(* Logix 5000 project; controller R5_CSS vendor 1 type 14 code 74 rev 19.11; software revision 19.01; part 19 of 20 *)
(* tags used below, declared in another part *)
   AlarmMasterDisable : BOOL;
   AutoTune : PIDE_AUTOTUNE;
   CSS_Heartbeat : BOOL;
   CSS_HeartbeatOffONS : BOOL;
   CSS_HeartbeatOnONS : BOOL;
   CSS_OK_TO_RUN : BOOL;   // PRU_RUN_DISABLE 0 = Cannot Run 1 = OK to Run
   CSS_Status_To_UTL_Comms : DINT;
   Fault : BOOL;
   FC101 : FLOW_CONTROL;   // QUENCH BASIN FLOW TRANSMITTER CONTROL
   FC101_Initialize : BOOL;
   FC101_Initialize_TON : TIMER;
   FT140_TOTAL_FLOW : REAL;
   LC101 : LEVEL_CONTROL;   // QUENCH TOWER BASIN LIT
   LC101_PIDE_AUTO : BOOL;
   LC101_PIDE_CV_Hold : REAL;
   LC303A : LEVEL_CONTROL;   // AQUEOUS PHASE OF PRIMARY SETTLER
   MSG_ConnectionRateSec : DINT;
   MSG_TimeoutMultiplier : DINT;
   MSG_UnconnectedTimeoutSec : DINT;
   PRU_Batch_Start : BOOL[32];
   PRU_Batch_Stop : BOOL[32];
   PRU_BatchNewID : DINT[10];
   PRU_BLOWER_SEQ : INT;   // PRU BLOWER SEQUENCE NUMBER
   PRU_MSG_CommsPath : MSG_CommsPath[9];
   PRU_MSG_Prefix : STRING;
   PRU_Quantity : DINT;
   PRU_SEQ_TMR : TIMER;   // PRU_SEQUENCE TIMER
   PRUA_Batch_Start_ONS : BOOL;
   PRUA_Batch_Stop_ONS : BOOL;
   PRUA_READ : INT[30];
   PRUA_READ_MSG : MESSAGE;
   PRUA_WRITE_MSG : MESSAGE;
   PRUB_Batch_Start_ONS : BOOL;
   PRUB_Batch_Stop_ONS : BOOL;
   PRUB_READ : INT[30];
   PRUB_READ_MSG : MESSAGE;
   PRUB_WRITE_MSG : MESSAGE;
   PRUC_Batch_Start_ONS : BOOL;
   PRUC_Batch_Stop_ONS : BOOL;
   PRUC_READ : INT[30];
   PRUC_READ_MSG : MESSAGE;
   PRUC_WRITE_MSG : MESSAGE;
   PRUD_Batch_Start_ONS : BOOL;
   PRUD_Batch_Stop_ONS : BOOL;
   PRUD_READ : INT[30];   // PRU D READ
   PRUD_READ_MSG : MESSAGE;
   PRUD_WRITE_MSG : MESSAGE;
   PRUE_Batch_Start_ONS : BOOL;
   PRUE_Batch_Stop_ONS : BOOL;
   PRUE_READ : INT[30];
   PRUE_READ_MSG : MESSAGE;
   PRUE_WRITE_MSG : MESSAGE;
   PRUF_Batch_Start_ONS : BOOL;
   PRUF_Batch_Stop_ONS : BOOL;
   PRUF_READ : INT[30];
   PRUF_READ_MSG : MESSAGE;
   PRUF_WRITE_MSG : MESSAGE;
   PRUG_Batch_Start_ONS : BOOL;
   PRUG_Batch_Stop_ONS : BOOL;
   PRUG_READ : INT[30];
   PRUG_READ_MSG : MESSAGE;
   PRUG_WRITE_MSG : MESSAGE;
   PRUH_Batch_Start_ONS : BOOL;
   PRUH_Batch_Stop_ONS : BOOL;
   PRUH_READ : INT[30];
   PRUH_READ_MSG : MESSAGE;
   PRUH_WRITE_MSG : MESSAGE;
   TestyBit : DINT;
   UTIL_1 : INT;   // ONE SHOTS FOR UTILITIES
   UTL_AlarmMaster : DINT;
   UTL_Comms : DINT[3];
   UTL_CommsLossAlm : BOOL;
   UTL_HeartbeatTimer : TIMER;
   UTL_READ_MSG : MESSAGE;
   WRS_OK : BOOL;
(* MainProgram, continued *)

ROUTINE TEMPORARY   (* ladder *)
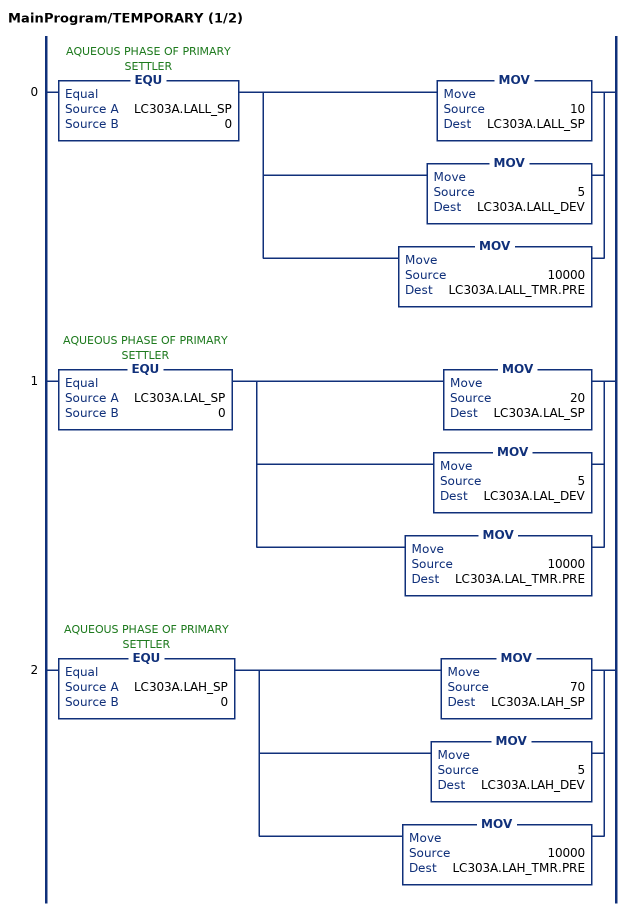
   0: EQU(LC303A.LALL_SP,0)[MOV(10,LC303A.LALL_SP) ,MOV(5,LC303A.LALL_DEV) ,MOV(10000,LC303A.LALL_TMR.PRE) ];
   1: EQU(LC303A.LAL_SP,0)[MOV(20,LC303A.LAL_SP) ,MOV(5,LC303A.LAL_DEV) ,MOV(10000,LC303A.LAL_TMR.PRE) ];
   2: EQU(LC303A.LAH_SP,0)[MOV(70,LC303A.LAH_SP) ,MOV(5,LC303A.LAH_DEV) ,MOV(10000,LC303A.LAH_TMR.PRE) ];
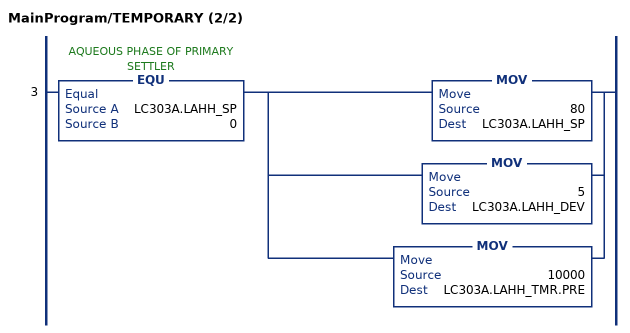
   3: EQU(LC303A.LAHH_SP,0)[MOV(80,LC303A.LAHH_SP) ,MOV(5,LC303A.LAHH_DEV) ,MOV(10000,LC303A.LAHH_TMR.PRE) ];
END_ROUTINE

ROUTINE UTIL   (* ladder *)
// UTILITIES LOGIC
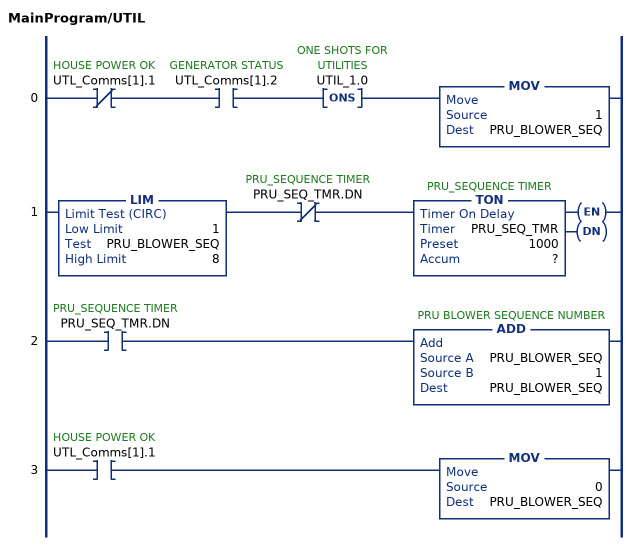
   0: XIO(UTL_Comms[1].1)XIC(UTL_Comms[1].2)ONS(UTIL_1.0)MOV(1,PRU_BLOWER_SEQ);
   1: LIM(1,PRU_BLOWER_SEQ,8)XIO(PRU_SEQ_TMR.DN)TON(PRU_SEQ_TMR,?,?);
   2: XIC(PRU_SEQ_TMR.DN)ADD(PRU_BLOWER_SEQ,1,PRU_BLOWER_SEQ);
   3: XIC(UTL_Comms[1].1)MOV(0,PRU_BLOWER_SEQ);
END_ROUTINE
END_PROGRAM

PROGRAM Never_Fault_Logic   (* main routine Main *)
VAR
   HMI_CONTROLLER_DISPLAY : MAJOR_FAULT := (TYPE := 3, CODE := 23);
   MAJORFAULT_RECORD : FAULTRECORD;
END_VAR

ROUTINE Main   (* ladder *)
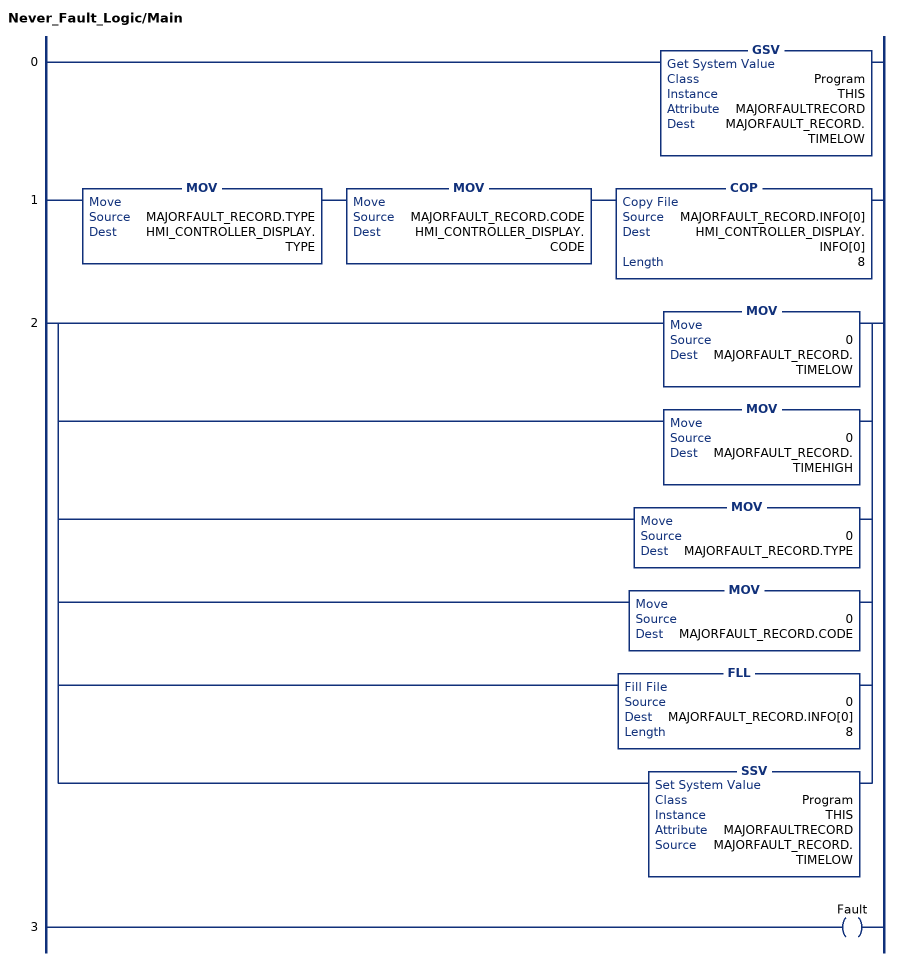
   0: GSV(Program,THIS,MAJORFAULTRECORD,MAJORFAULT_RECORD.TIMELOW);
   1: MOV(MAJORFAULT_RECORD.TYPE,HMI_CONTROLLER_DISPLAY.TYPE)MOV(MAJORFAULT_RECORD.CODE,HMI_CONTROLLER_DISPLAY.CODE)COP(MAJORFAULT_RECORD.INFO[0],HMI_CONTROLLER_DISPLAY.INFO[0],8);
   2: [MOV(0,MAJORFAULT_RECORD.TIMELOW) ,MOV(0,MAJORFAULT_RECORD.TIMEHIGH) ,MOV(0,MAJORFAULT_RECORD.TYPE) ,MOV(0,MAJORFAULT_RECORD.CODE) ,FLL(0,MAJORFAULT_RECORD.INFO[0],8) ,SSV(Program,THIS,MAJORFAULTRECORD,MAJORFAULT_RECORD.TIMELOW) ];
   3: OTE(Fault);
END_ROUTINE
END_PROGRAM

PROGRAM PIDE   (* main routine Main *)
VAR
   BNOT_01 : FBD_BOOLEAN_NOT := (Out := 1);
   BNOT_02 : FBD_BOOLEAN_NOT := (In := 1);
   SUB_01 : FBD_MATH := (SourceA := 1.4874992, SourceB := 30.0, Dest := -28.5125);
END_VAR

ROUTINE LC101   (* function block diagram *)
   SHEET 1
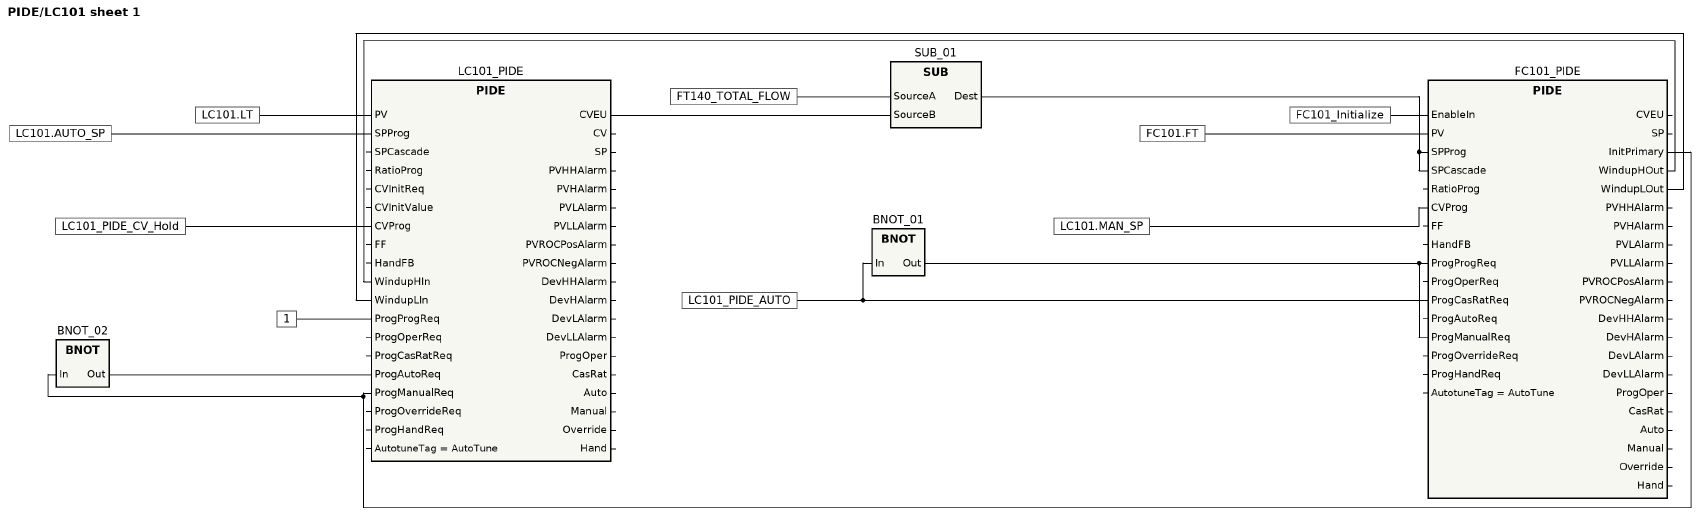
   BNOT_02 : BNOT(In := FC101_PIDE.InitPrimary {feedback});
   LC101_PIDE : PIDE(PV := LC101.LT, SPProg := LC101.AUTO_SP, CVProg := LC101_PIDE_CV_Hold, WindupHIn := FC101_PIDE.WindupHOut {feedback}, WindupLIn := FC101_PIDE.WindupLOut {feedback}, ProgProgReq := 1, ProgAutoReq := BNOT_02.Out, ProgManualReq := FC101_PIDE.InitPrimary {feedback}, AutotuneTag := AutoTune);   // unwired pins: SPCascade RatioProg CVInitReq CVInitValue FF HandFB ProgOperReq ProgCasRatReq ProgOverrideReq ProgHandReq CV SP PVHHAlarm PVHAlarm PVLAlarm PVLLAlarm PVROCPosAlarm PVROCNegAlarm DevHHAlarm DevHAlarm DevLAlarm DevLLAlarm ProgOper CasRat Auto Manual Override Hand
   BNOT_01 : BNOT(In := LC101_PIDE_AUTO);
   SUB_01 : SUB(SourceA := FT140_TOTAL_FLOW, SourceB := LC101_PIDE.CVEU);
   FC101_PIDE : PIDE(EnableIn := FC101_Initialize, PV := FC101.FT, SPProg := SUB_01.Dest, SPCascade := SUB_01.Dest, CVProg := LC101.MAN_SP, ProgProgReq := BNOT_01.Out, ProgCasRatReq := LC101_PIDE_AUTO, ProgManualReq := BNOT_01.Out, AutotuneTag := AutoTune);   // unwired pins: RatioProg FF HandFB ProgOperReq ProgAutoReq ProgOverrideReq ProgHandReq CVEU SP PVHHAlarm PVHAlarm PVLAlarm PVLLAlarm PVROCPosAlarm PVROCNegAlarm DevHHAlarm DevHAlarm DevLAlarm DevLLAlarm ProgOper CasRat Auto Manual Override Hand
END_ROUTINE

ROUTINE Main   (* ladder *)
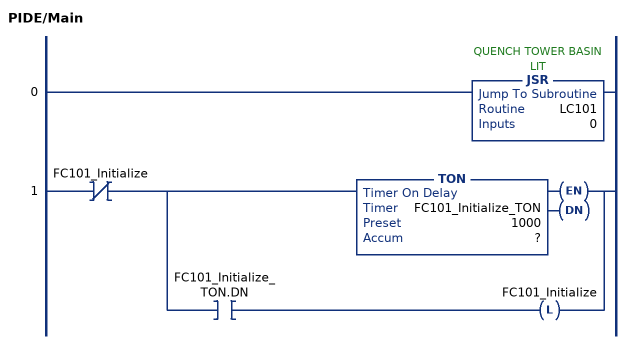
   0: JSR(LC101,0);
   1: XIO(FC101_Initialize)[TON(FC101_Initialize_TON,?,?) ,XIC(FC101_Initialize_TON.DN) OTL(FC101_Initialize) ];
END_ROUTINE
END_PROGRAM

PROGRAM POD1_MSG   (* main routine MSG *)
VAR
   PRU_BatchNewID_old : DINT[5];
END_VAR

ROUTINE MSG   (* ladder *)
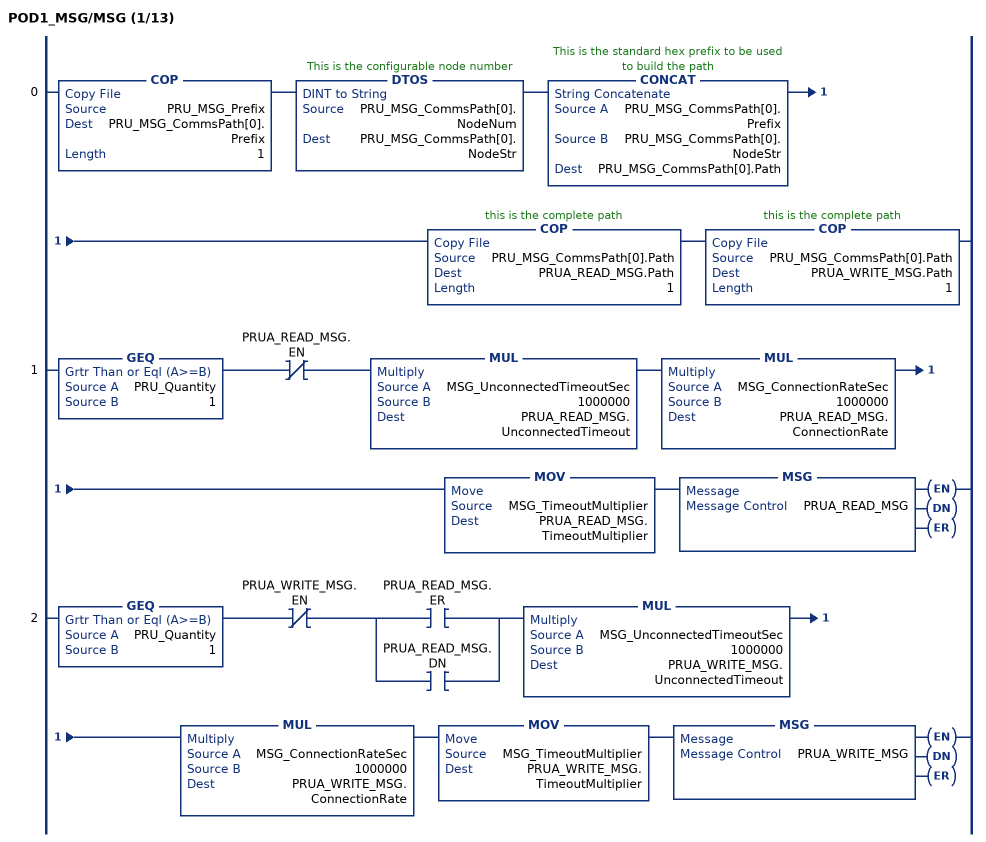
   0: COP(PRU_MSG_Prefix,PRU_MSG_CommsPath[0].Prefix,1)DTOS(PRU_MSG_CommsPath[0].NodeNum,PRU_MSG_CommsPath[0].NodeStr)CONCAT(PRU_MSG_CommsPath[0].Prefix,PRU_MSG_CommsPath[0].NodeStr,PRU_MSG_CommsPath[0].Path)COP(PRU_MSG_CommsPath[0].Path,PRUA_READ_MSG.Path,1)COP(PRU_MSG_CommsPath[0].Path,PRUA_WRITE_MSG.Path,1);
   1: GEQ(PRU_Quantity,1)XIO(PRUA_READ_MSG.EN)MUL(MSG_UnconnectedTimeoutSec,1000000,PRUA_READ_MSG.UnconnectedTimeout)MUL(MSG_ConnectionRateSec,1000000,PRUA_READ_MSG.ConnectionRate)MOV(MSG_TimeoutMultiplier,PRUA_READ_MSG.TimeoutMultiplier)MSG(PRUA_READ_MSG);
   2: GEQ(PRU_Quantity,1)XIO(PRUA_WRITE_MSG.EN)[XIC(PRUA_READ_MSG.ER) ,XIC(PRUA_READ_MSG.DN) ]MUL(MSG_UnconnectedTimeoutSec,1000000,PRUA_WRITE_MSG.UnconnectedTimeout)MUL(MSG_ConnectionRateSec,1000000,PRUA_WRITE_MSG.ConnectionRate)MOV(MSG_TimeoutMultiplier,PRUA_WRITE_MSG.TimeoutMultiplier)MSG(PRUA_WRITE_MSG);
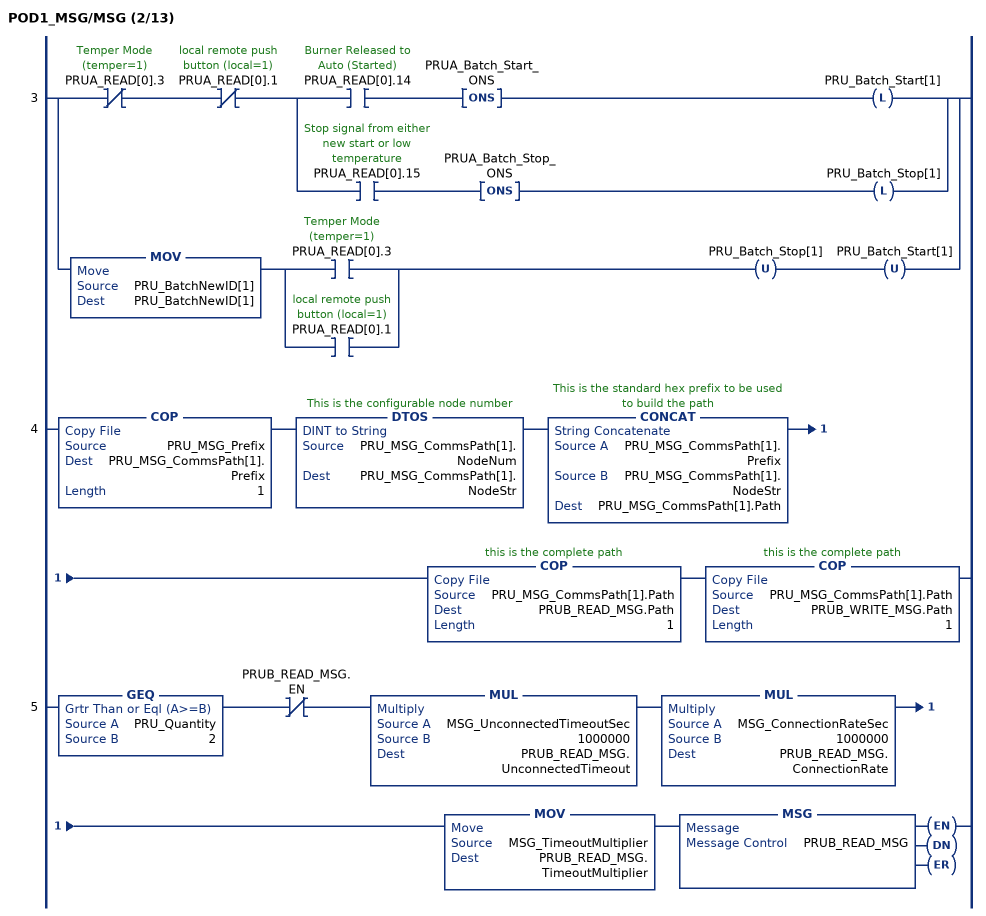
   3: [XIO(PRUA_READ[0].3) XIO(PRUA_READ[0].1) [XIC(PRUA_READ[0].14) ONS(PRUA_Batch_Start_ONS) OTL(PRU_Batch_Start[1]) ,XIC(PRUA_READ[0].15) ONS(PRUA_Batch_Stop_ONS) OTL(PRU_Batch_Stop[1]) ] ,MOV(PRU_BatchNewID[1],PRU_BatchNewID[1]) [XIC(PRUA_READ[0].3) ,XIC(PRUA_READ[0].1) ] OTU(PRU_Batch_Stop[1]) OTU(PRU_Batch_Start[1]) ];
   4: COP(PRU_MSG_Prefix,PRU_MSG_CommsPath[1].Prefix,1)DTOS(PRU_MSG_CommsPath[1].NodeNum,PRU_MSG_CommsPath[1].NodeStr)CONCAT(PRU_MSG_CommsPath[1].Prefix,PRU_MSG_CommsPath[1].NodeStr,PRU_MSG_CommsPath[1].Path)COP(PRU_MSG_CommsPath[1].Path,PRUB_READ_MSG.Path,1)COP(PRU_MSG_CommsPath[1].Path,PRUB_WRITE_MSG.Path,1);
   5: GEQ(PRU_Quantity,2)XIO(PRUB_READ_MSG.EN)MUL(MSG_UnconnectedTimeoutSec,1000000,PRUB_READ_MSG.UnconnectedTimeout)MUL(MSG_ConnectionRateSec,1000000,PRUB_READ_MSG.ConnectionRate)MOV(MSG_TimeoutMultiplier,PRUB_READ_MSG.TimeoutMultiplier)MSG(PRUB_READ_MSG);
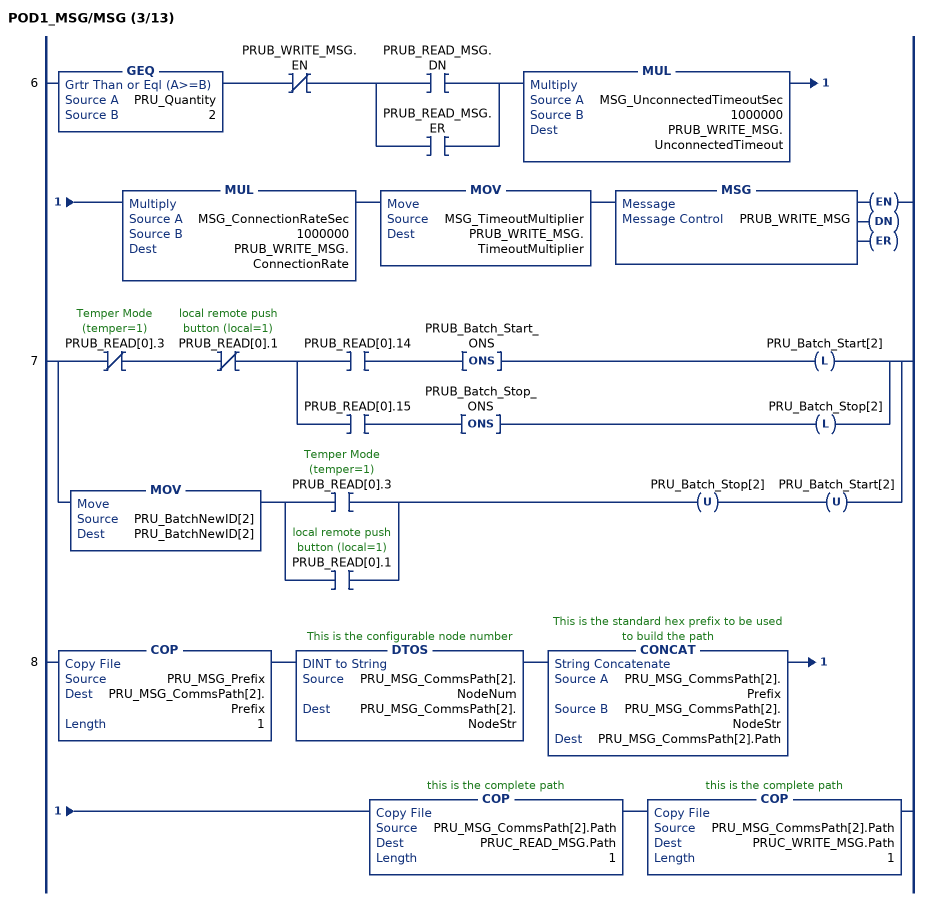
   6: GEQ(PRU_Quantity,2)XIO(PRUB_WRITE_MSG.EN)[XIC(PRUB_READ_MSG.DN) ,XIC(PRUB_READ_MSG.ER) ]MUL(MSG_UnconnectedTimeoutSec,1000000,PRUB_WRITE_MSG.UnconnectedTimeout)MUL(MSG_ConnectionRateSec,1000000,PRUB_WRITE_MSG.ConnectionRate)MOV(MSG_TimeoutMultiplier,PRUB_WRITE_MSG.TimeoutMultiplier)MSG(PRUB_WRITE_MSG);
   7: [XIO(PRUB_READ[0].3) XIO(PRUB_READ[0].1) [XIC(PRUB_READ[0].14) ONS(PRUB_Batch_Start_ONS) OTL(PRU_Batch_Start[2]) ,XIC(PRUB_READ[0].15) ONS(PRUB_Batch_Stop_ONS) OTL(PRU_Batch_Stop[2]) ] ,MOV(PRU_BatchNewID[2],PRU_BatchNewID[2]) [XIC(PRUB_READ[0].3) ,XIC(PRUB_READ[0].1) ] OTU(PRU_Batch_Stop[2]) OTU(PRU_Batch_Start[2]) ];
   8: COP(PRU_MSG_Prefix,PRU_MSG_CommsPath[2].Prefix,1)DTOS(PRU_MSG_CommsPath[2].NodeNum,PRU_MSG_CommsPath[2].NodeStr)CONCAT(PRU_MSG_CommsPath[2].Prefix,PRU_MSG_CommsPath[2].NodeStr,PRU_MSG_CommsPath[2].Path)COP(PRU_MSG_CommsPath[2].Path,PRUC_READ_MSG.Path,1)COP(PRU_MSG_CommsPath[2].Path,PRUC_WRITE_MSG.Path,1);
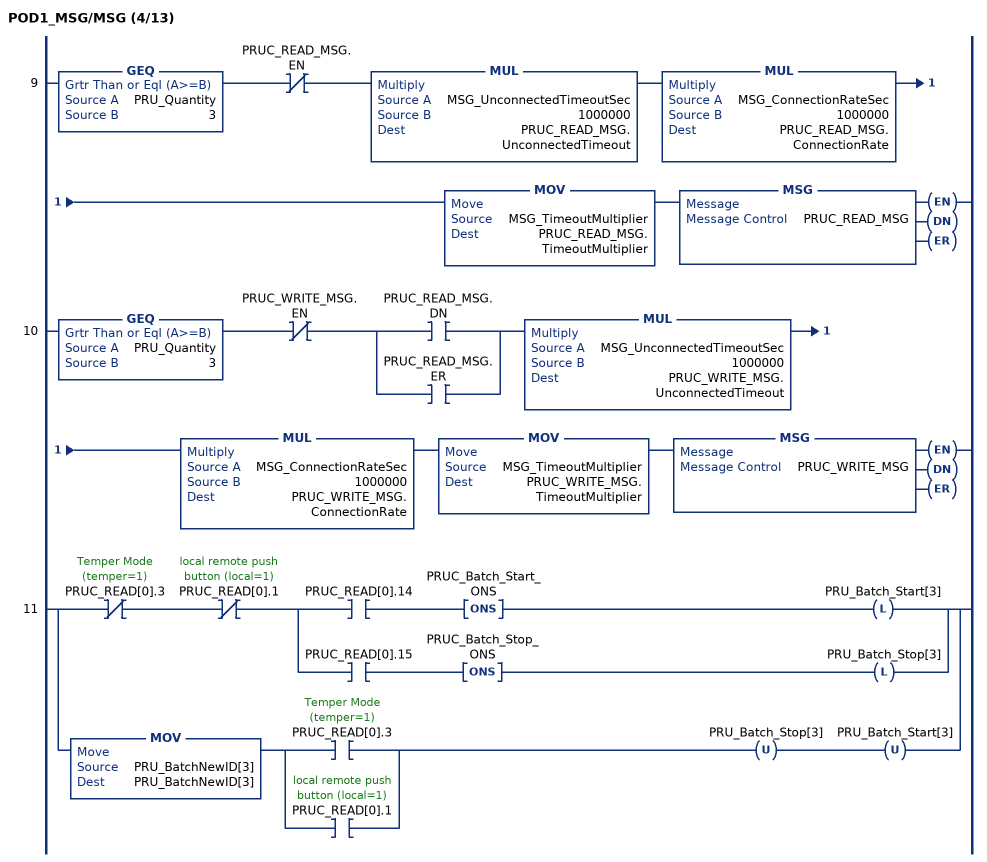
   9: GEQ(PRU_Quantity,3)XIO(PRUC_READ_MSG.EN)MUL(MSG_UnconnectedTimeoutSec,1000000,PRUC_READ_MSG.UnconnectedTimeout)MUL(MSG_ConnectionRateSec,1000000,PRUC_READ_MSG.ConnectionRate)MOV(MSG_TimeoutMultiplier,PRUC_READ_MSG.TimeoutMultiplier)MSG(PRUC_READ_MSG);
   10: GEQ(PRU_Quantity,3)XIO(PRUC_WRITE_MSG.EN)[XIC(PRUC_READ_MSG.DN) ,XIC(PRUC_READ_MSG.ER) ]MUL(MSG_UnconnectedTimeoutSec,1000000,PRUC_WRITE_MSG.UnconnectedTimeout)MUL(MSG_ConnectionRateSec,1000000,PRUC_WRITE_MSG.ConnectionRate)MOV(MSG_TimeoutMultiplier,PRUC_WRITE_MSG.TimeoutMultiplier)MSG(PRUC_WRITE_MSG);
   11: [XIO(PRUC_READ[0].3) XIO(PRUC_READ[0].1) [XIC(PRUC_READ[0].14) ONS(PRUC_Batch_Start_ONS) OTL(PRU_Batch_Start[3]) ,XIC(PRUC_READ[0].15) ONS(PRUC_Batch_Stop_ONS) OTL(PRU_Batch_Stop[3]) ] ,MOV(PRU_BatchNewID[3],PRU_BatchNewID[3]) [XIC(PRUC_READ[0].3) ,XIC(PRUC_READ[0].1) ] OTU(PRU_Batch_Stop[3]) OTU(PRU_Batch_Start[3]) ];
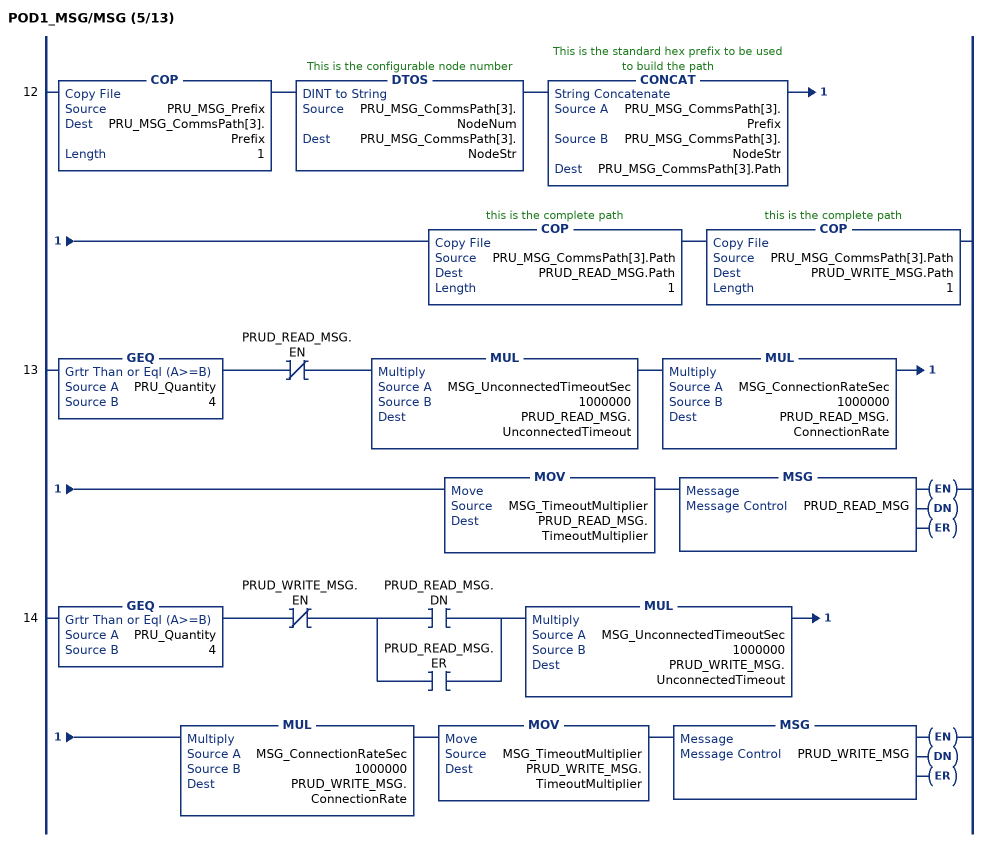
   12: COP(PRU_MSG_Prefix,PRU_MSG_CommsPath[3].Prefix,1)DTOS(PRU_MSG_CommsPath[3].NodeNum,PRU_MSG_CommsPath[3].NodeStr)CONCAT(PRU_MSG_CommsPath[3].Prefix,PRU_MSG_CommsPath[3].NodeStr,PRU_MSG_CommsPath[3].Path)COP(PRU_MSG_CommsPath[3].Path,PRUD_READ_MSG.Path,1)COP(PRU_MSG_CommsPath[3].Path,PRUD_WRITE_MSG.Path,1);
   13: GEQ(PRU_Quantity,4)XIO(PRUD_READ_MSG.EN)MUL(MSG_UnconnectedTimeoutSec,1000000,PRUD_READ_MSG.UnconnectedTimeout)MUL(MSG_ConnectionRateSec,1000000,PRUD_READ_MSG.ConnectionRate)MOV(MSG_TimeoutMultiplier,PRUD_READ_MSG.TimeoutMultiplier)MSG(PRUD_READ_MSG);
   14: GEQ(PRU_Quantity,4)XIO(PRUD_WRITE_MSG.EN)[XIC(PRUD_READ_MSG.DN) ,XIC(PRUD_READ_MSG.ER) ]MUL(MSG_UnconnectedTimeoutSec,1000000,PRUD_WRITE_MSG.UnconnectedTimeout)MUL(MSG_ConnectionRateSec,1000000,PRUD_WRITE_MSG.ConnectionRate)MOV(MSG_TimeoutMultiplier,PRUD_WRITE_MSG.TimeoutMultiplier)MSG(PRUD_WRITE_MSG);
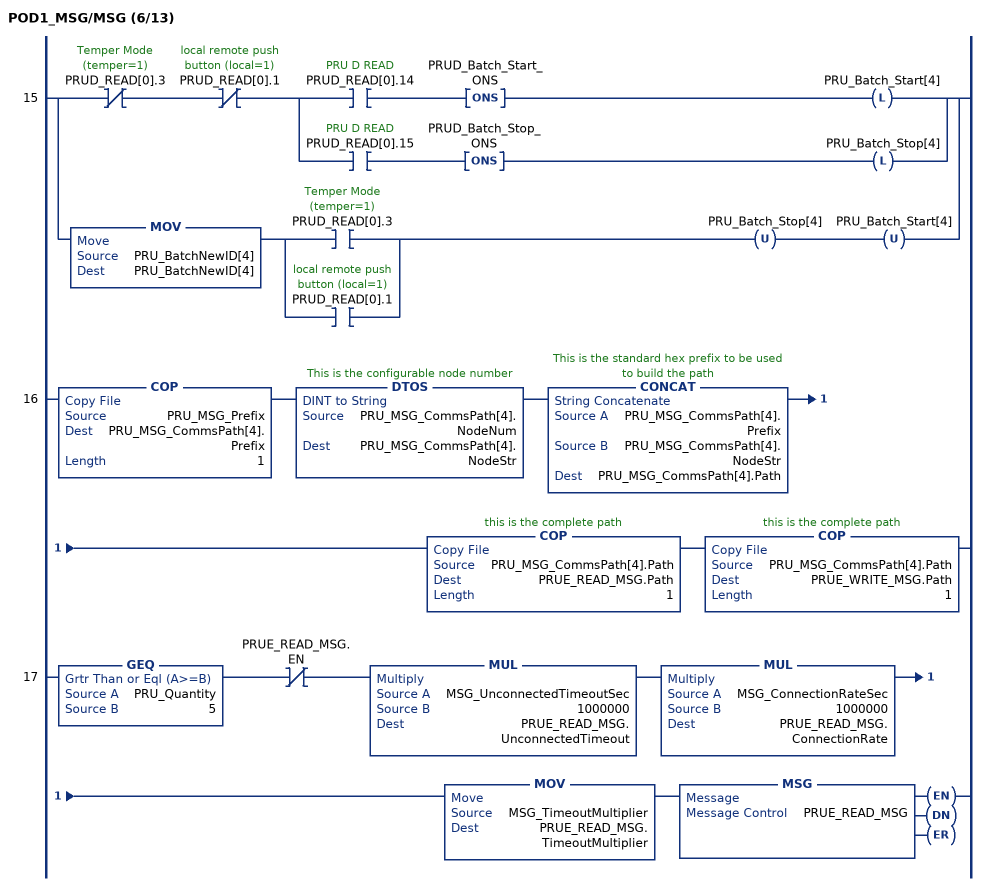
   15: [XIO(PRUD_READ[0].3) XIO(PRUD_READ[0].1) [XIC(PRUD_READ[0].14) ONS(PRUD_Batch_Start_ONS) OTL(PRU_Batch_Start[4]) ,XIC(PRUD_READ[0].15) ONS(PRUD_Batch_Stop_ONS) OTL(PRU_Batch_Stop[4]) ] ,MOV(PRU_BatchNewID[4],PRU_BatchNewID[4]) [XIC(PRUD_READ[0].3) ,XIC(PRUD_READ[0].1) ] OTU(PRU_Batch_Stop[4]) OTU(PRU_Batch_Start[4]) ];
   16: COP(PRU_MSG_Prefix,PRU_MSG_CommsPath[4].Prefix,1)DTOS(PRU_MSG_CommsPath[4].NodeNum,PRU_MSG_CommsPath[4].NodeStr)CONCAT(PRU_MSG_CommsPath[4].Prefix,PRU_MSG_CommsPath[4].NodeStr,PRU_MSG_CommsPath[4].Path)COP(PRU_MSG_CommsPath[4].Path,PRUE_READ_MSG.Path,1)COP(PRU_MSG_CommsPath[4].Path,PRUE_WRITE_MSG.Path,1);
   17: GEQ(PRU_Quantity,5)XIO(PRUE_READ_MSG.EN)MUL(MSG_UnconnectedTimeoutSec,1000000,PRUE_READ_MSG.UnconnectedTimeout)MUL(MSG_ConnectionRateSec,1000000,PRUE_READ_MSG.ConnectionRate)MOV(MSG_TimeoutMultiplier,PRUE_READ_MSG.TimeoutMultiplier)MSG(PRUE_READ_MSG);
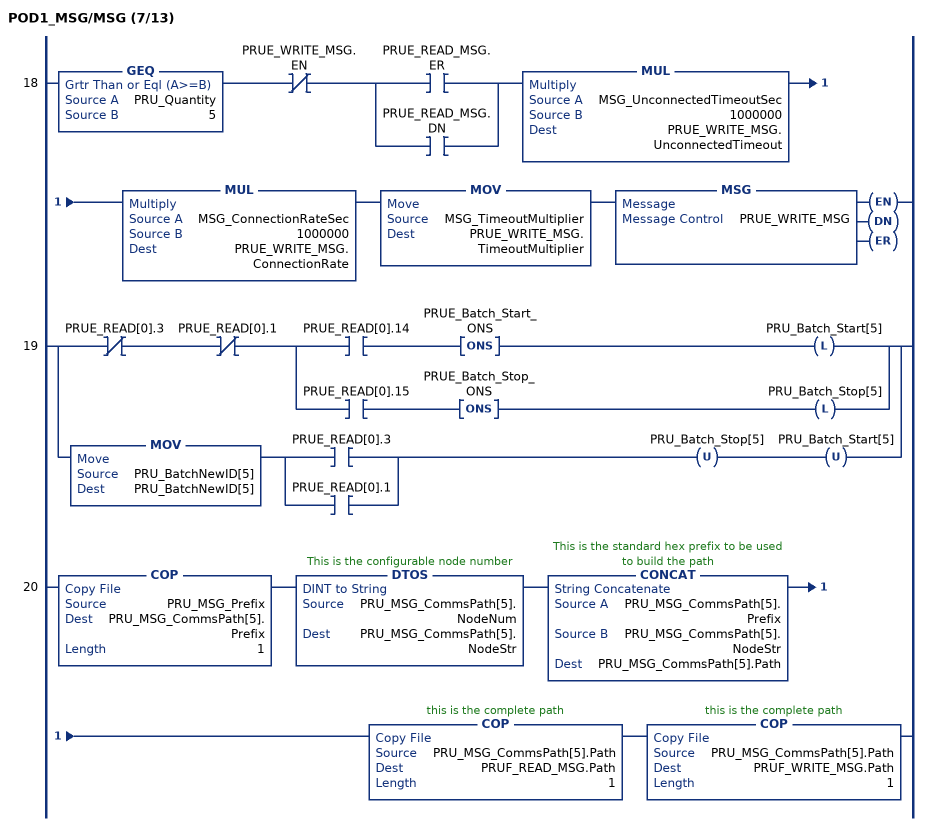
   18: GEQ(PRU_Quantity,5)XIO(PRUE_WRITE_MSG.EN)[XIC(PRUE_READ_MSG.ER) ,XIC(PRUE_READ_MSG.DN) ]MUL(MSG_UnconnectedTimeoutSec,1000000,PRUE_WRITE_MSG.UnconnectedTimeout)MUL(MSG_ConnectionRateSec,1000000,PRUE_WRITE_MSG.ConnectionRate)MOV(MSG_TimeoutMultiplier,PRUE_WRITE_MSG.TimeoutMultiplier)MSG(PRUE_WRITE_MSG);
   19: [XIO(PRUE_READ[0].3) XIO(PRUE_READ[0].1) [XIC(PRUE_READ[0].14) ONS(PRUE_Batch_Start_ONS) OTL(PRU_Batch_Start[5]) ,XIC(PRUE_READ[0].15) ONS(PRUE_Batch_Stop_ONS) OTL(PRU_Batch_Stop[5]) ] ,MOV(PRU_BatchNewID[5],PRU_BatchNewID[5]) [XIC(PRUE_READ[0].3) ,XIC(PRUE_READ[0].1) ] OTU(PRU_Batch_Stop[5]) OTU(PRU_Batch_Start[5]) ];
   20: COP(PRU_MSG_Prefix,PRU_MSG_CommsPath[5].Prefix,1)DTOS(PRU_MSG_CommsPath[5].NodeNum,PRU_MSG_CommsPath[5].NodeStr)CONCAT(PRU_MSG_CommsPath[5].Prefix,PRU_MSG_CommsPath[5].NodeStr,PRU_MSG_CommsPath[5].Path)COP(PRU_MSG_CommsPath[5].Path,PRUF_READ_MSG.Path,1)COP(PRU_MSG_CommsPath[5].Path,PRUF_WRITE_MSG.Path,1);
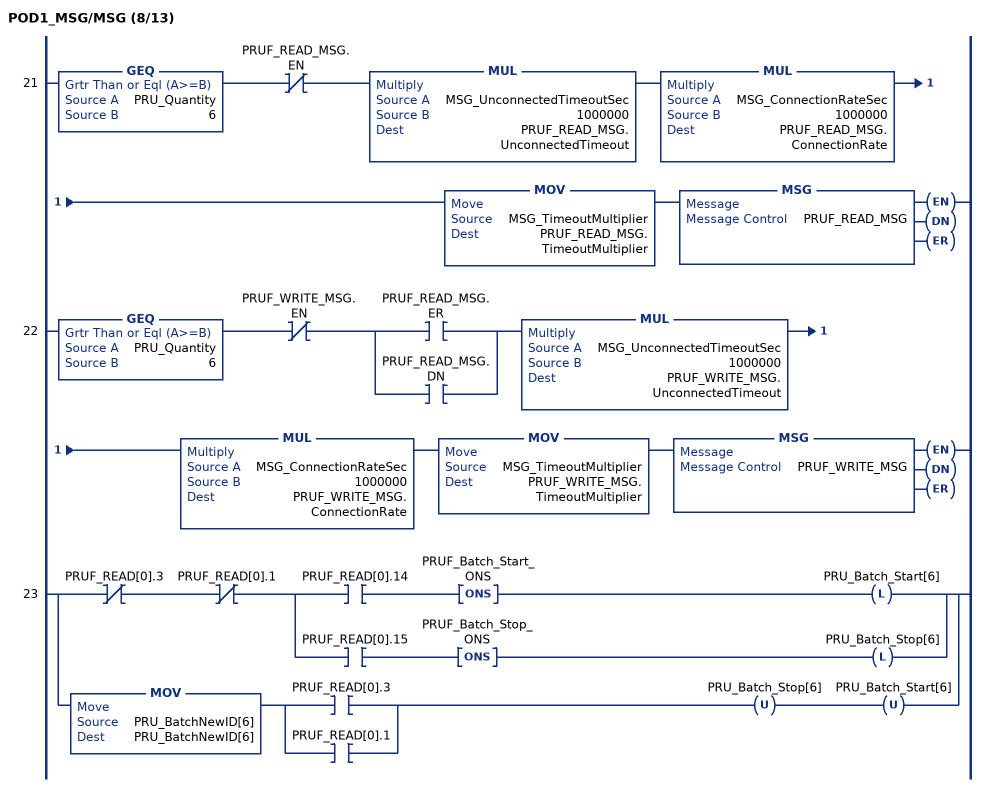
   21: GEQ(PRU_Quantity,6)XIO(PRUF_READ_MSG.EN)MUL(MSG_UnconnectedTimeoutSec,1000000,PRUF_READ_MSG.UnconnectedTimeout)MUL(MSG_ConnectionRateSec,1000000,PRUF_READ_MSG.ConnectionRate)MOV(MSG_TimeoutMultiplier,PRUF_READ_MSG.TimeoutMultiplier)MSG(PRUF_READ_MSG);
   22: GEQ(PRU_Quantity,6)XIO(PRUF_WRITE_MSG.EN)[XIC(PRUF_READ_MSG.ER) ,XIC(PRUF_READ_MSG.DN) ]MUL(MSG_UnconnectedTimeoutSec,1000000,PRUF_WRITE_MSG.UnconnectedTimeout)MUL(MSG_ConnectionRateSec,1000000,PRUF_WRITE_MSG.ConnectionRate)MOV(MSG_TimeoutMultiplier,PRUF_WRITE_MSG.TimeoutMultiplier)MSG(PRUF_WRITE_MSG);
   23: [XIO(PRUF_READ[0].3) XIO(PRUF_READ[0].1) [XIC(PRUF_READ[0].14) ONS(PRUF_Batch_Start_ONS) OTL(PRU_Batch_Start[6]) ,XIC(PRUF_READ[0].15) ONS(PRUF_Batch_Stop_ONS) OTL(PRU_Batch_Stop[6]) ] ,MOV(PRU_BatchNewID[6],PRU_BatchNewID[6]) [XIC(PRUF_READ[0].3) ,XIC(PRUF_READ[0].1) ] OTU(PRU_Batch_Stop[6]) OTU(PRU_Batch_Start[6]) ];
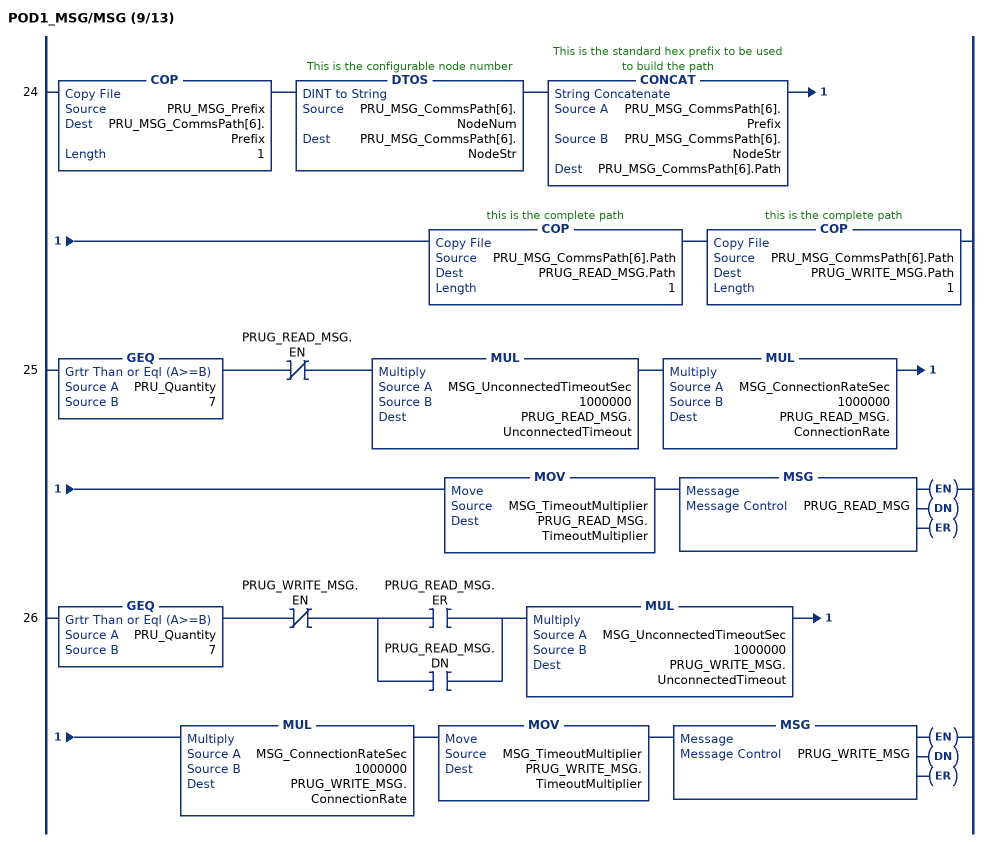
   24: COP(PRU_MSG_Prefix,PRU_MSG_CommsPath[6].Prefix,1)DTOS(PRU_MSG_CommsPath[6].NodeNum,PRU_MSG_CommsPath[6].NodeStr)CONCAT(PRU_MSG_CommsPath[6].Prefix,PRU_MSG_CommsPath[6].NodeStr,PRU_MSG_CommsPath[6].Path)COP(PRU_MSG_CommsPath[6].Path,PRUG_READ_MSG.Path,1)COP(PRU_MSG_CommsPath[6].Path,PRUG_WRITE_MSG.Path,1);
   25: GEQ(PRU_Quantity,7)XIO(PRUG_READ_MSG.EN)MUL(MSG_UnconnectedTimeoutSec,1000000,PRUG_READ_MSG.UnconnectedTimeout)MUL(MSG_ConnectionRateSec,1000000,PRUG_READ_MSG.ConnectionRate)MOV(MSG_TimeoutMultiplier,PRUG_READ_MSG.TimeoutMultiplier)MSG(PRUG_READ_MSG);
   26: GEQ(PRU_Quantity,7)XIO(PRUG_WRITE_MSG.EN)[XIC(PRUG_READ_MSG.ER) ,XIC(PRUG_READ_MSG.DN) ]MUL(MSG_UnconnectedTimeoutSec,1000000,PRUG_WRITE_MSG.UnconnectedTimeout)MUL(MSG_ConnectionRateSec,1000000,PRUG_WRITE_MSG.ConnectionRate)MOV(MSG_TimeoutMultiplier,PRUG_WRITE_MSG.TimeoutMultiplier)MSG(PRUG_WRITE_MSG);
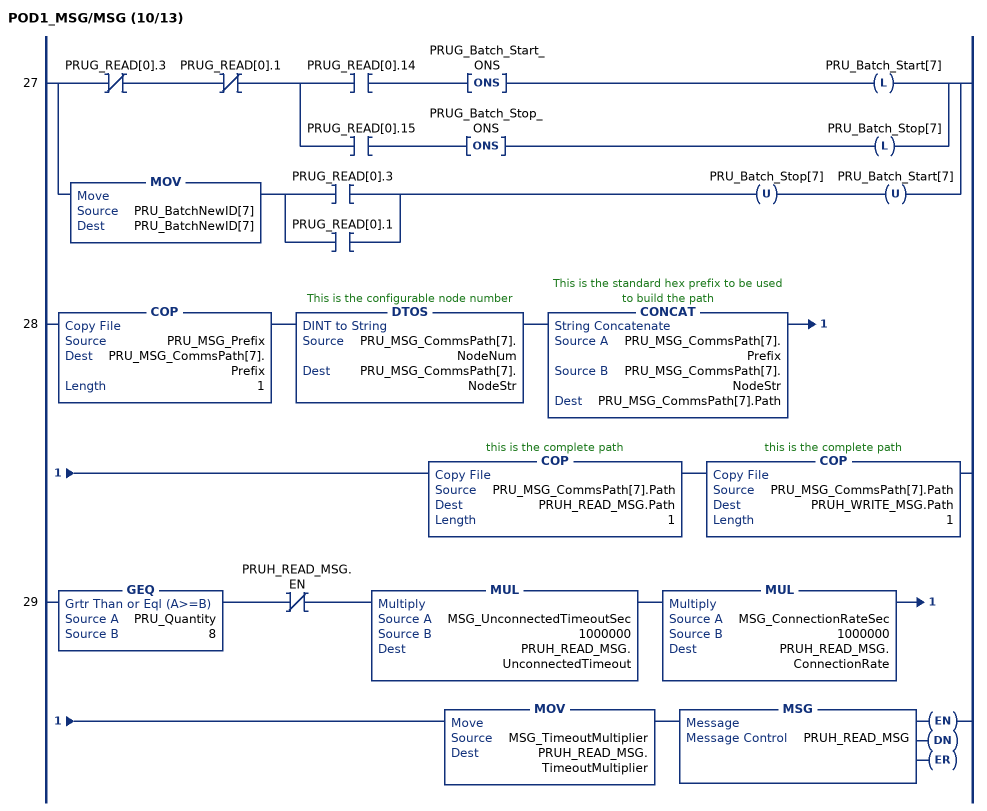
   27: [XIO(PRUG_READ[0].3) XIO(PRUG_READ[0].1) [XIC(PRUG_READ[0].14) ONS(PRUG_Batch_Start_ONS) OTL(PRU_Batch_Start[7]) ,XIC(PRUG_READ[0].15) ONS(PRUG_Batch_Stop_ONS) OTL(PRU_Batch_Stop[7]) ] ,MOV(PRU_BatchNewID[7],PRU_BatchNewID[7]) [XIC(PRUG_READ[0].3) ,XIC(PRUG_READ[0].1) ] OTU(PRU_Batch_Stop[7]) OTU(PRU_Batch_Start[7]) ];
   28: COP(PRU_MSG_Prefix,PRU_MSG_CommsPath[7].Prefix,1)DTOS(PRU_MSG_CommsPath[7].NodeNum,PRU_MSG_CommsPath[7].NodeStr)CONCAT(PRU_MSG_CommsPath[7].Prefix,PRU_MSG_CommsPath[7].NodeStr,PRU_MSG_CommsPath[7].Path)COP(PRU_MSG_CommsPath[7].Path,PRUH_READ_MSG.Path,1)COP(PRU_MSG_CommsPath[7].Path,PRUH_WRITE_MSG.Path,1);
   29: GEQ(PRU_Quantity,8)XIO(PRUH_READ_MSG.EN)MUL(MSG_UnconnectedTimeoutSec,1000000,PRUH_READ_MSG.UnconnectedTimeout)MUL(MSG_ConnectionRateSec,1000000,PRUH_READ_MSG.ConnectionRate)MOV(MSG_TimeoutMultiplier,PRUH_READ_MSG.TimeoutMultiplier)MSG(PRUH_READ_MSG);
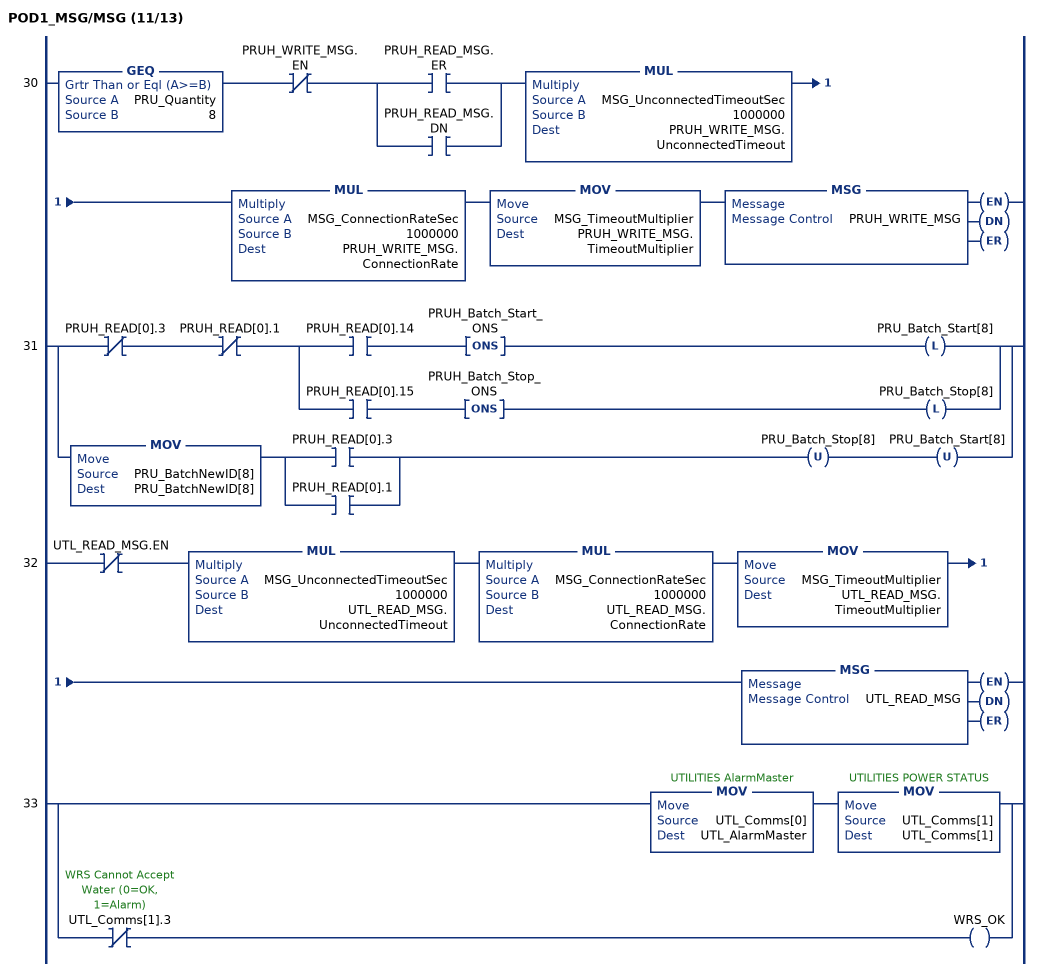
   30: GEQ(PRU_Quantity,8)XIO(PRUH_WRITE_MSG.EN)[XIC(PRUH_READ_MSG.ER) ,XIC(PRUH_READ_MSG.DN) ]MUL(MSG_UnconnectedTimeoutSec,1000000,PRUH_WRITE_MSG.UnconnectedTimeout)MUL(MSG_ConnectionRateSec,1000000,PRUH_WRITE_MSG.ConnectionRate)MOV(MSG_TimeoutMultiplier,PRUH_WRITE_MSG.TimeoutMultiplier)MSG(PRUH_WRITE_MSG);
   31: [XIO(PRUH_READ[0].3) XIO(PRUH_READ[0].1) [XIC(PRUH_READ[0].14) ONS(PRUH_Batch_Start_ONS) OTL(PRU_Batch_Start[8]) ,XIC(PRUH_READ[0].15) ONS(PRUH_Batch_Stop_ONS) OTL(PRU_Batch_Stop[8]) ] ,MOV(PRU_BatchNewID[8],PRU_BatchNewID[8]) [XIC(PRUH_READ[0].3) ,XIC(PRUH_READ[0].1) ] OTU(PRU_Batch_Stop[8]) OTU(PRU_Batch_Start[8]) ];
   32: XIO(UTL_READ_MSG.EN)MUL(MSG_UnconnectedTimeoutSec,1000000,UTL_READ_MSG.UnconnectedTimeout)MUL(MSG_ConnectionRateSec,1000000,UTL_READ_MSG.ConnectionRate)MOV(MSG_TimeoutMultiplier,UTL_READ_MSG.TimeoutMultiplier)MSG(UTL_READ_MSG);
   33: [MOV(UTL_Comms[0],UTL_AlarmMaster) MOV(UTL_Comms[1],UTL_Comms[1]) ,XIO(UTL_Comms[1].3) OTE(WRS_OK) ];
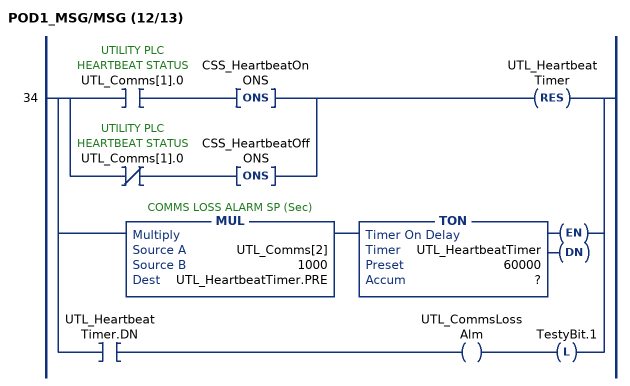
   34: [[XIC(UTL_Comms[1].0) ONS(CSS_HeartbeatOnONS) ,XIO(UTL_Comms[1].0) ONS(CSS_HeartbeatOffONS) ] RES(UTL_HeartbeatTimer) ,MUL(UTL_Comms[2],1000,UTL_HeartbeatTimer.PRE) TON(UTL_HeartbeatTimer,?,?) ,XIC(UTL_HeartbeatTimer.DN) OTE(UTL_CommsLossAlm) OTL(TestyBit.1) ];
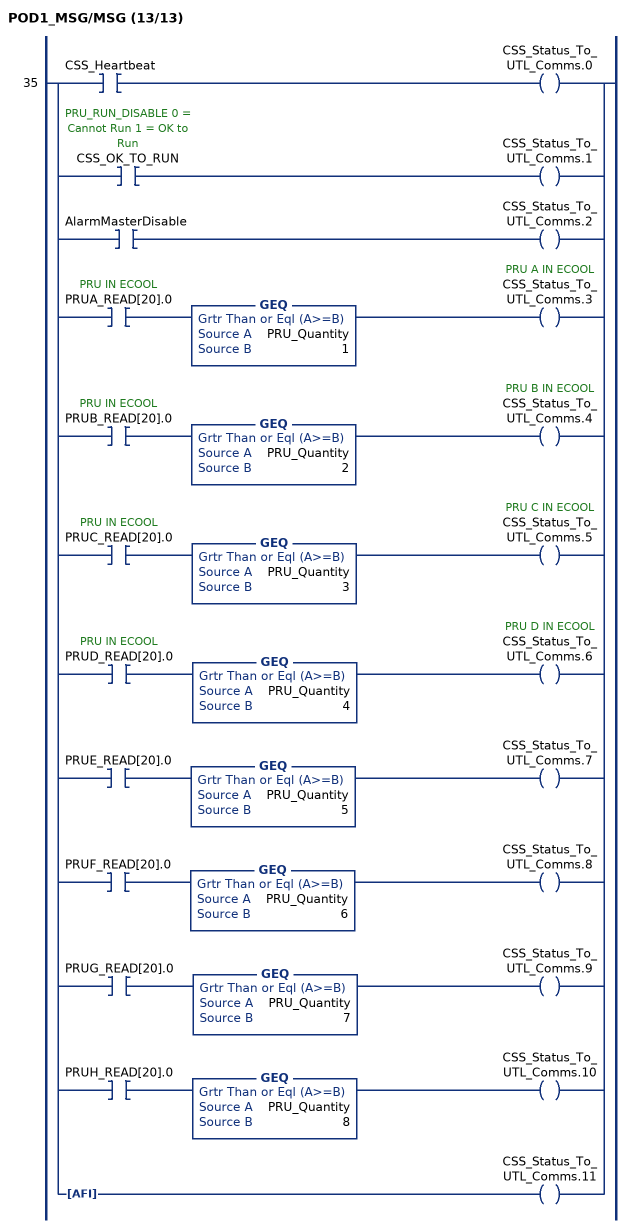
   35: [XIC(CSS_Heartbeat) OTE(CSS_Status_To_UTL_Comms.0) ,XIC(CSS_OK_TO_RUN) OTE(CSS_Status_To_UTL_Comms.1) ,XIC(AlarmMasterDisable) OTE(CSS_Status_To_UTL_Comms.2) ,XIC(PRUA_READ[20].0) GEQ(PRU_Quantity,1) OTE(CSS_Status_To_UTL_Comms.3) ,XIC(PRUB_READ[20].0) GEQ(PRU_Quantity,2) OTE(CSS_Status_To_UTL_Comms.4) ,XIC(PRUC_READ[20].0) GEQ(PRU_Quantity,3) OTE(CSS_Status_To_UTL_Comms.5) ,XIC(PRUD_READ[20].0) GEQ(PRU_Quantity,4) OTE(CSS_Status_To_UTL_Comms.6) ,XIC(PRUE_READ[20].0) GEQ(PRU_Quantity,5) OTE(CSS_Status_To_UTL_Comms.7) ,XIC(PRUF_READ[20].0) GEQ(PRU_Quantity,6) OTE(CSS_Status_To_UTL_Comms.8) ,XIC(PRUG_READ[20].0) GEQ(PRU_Quantity,7) OTE(CSS_Status_To_UTL_Comms.9) ,XIC(PRUH_READ[20].0) GEQ(PRU_Quantity,8) OTE(CSS_Status_To_UTL_Comms.10) ,AFI() OTE(CSS_Status_To_UTL_Comms.11) ];
END_ROUTINE
END_PROGRAM
